# EPICS substitutions: ek9000App/Db/EL7047.substitutions
file EL7047.template
{       pattern
        {
                TERMINAL,

        }
        {
        }
}
